{attribute 'qualified_only'}
{attribute 'strict'}
{attribute 'to_string'}
TYPE SkillCommand :
(
	KEINE		:= 0,
	STARTEN		:= 1,
	STOPPEN		:= 2,
	RESETTEN 	:= 3
);
END_TYPE

(* stored: Version 1.1.0.1
   DUT SkillCommand: Id {58c5248f-54d1-462d-851b-c21f37b367a1} *)
